// TIA Portal V18 export
TYPE "PLCtoMES_ResultsStoredScanExchange_ext"
// stored: IsFailsafeCompliant false
   STRUCT
      Load_Scanner1ChickInReq : Bool;   // Scanner1查询
      Load_Scanner2ChickInReq : Bool;   // Spare
      Load_Scanner3ChickInReq : Bool;   // Spare
      Load_Scanner4ChickInReq : Bool;   // Spare
      Load_Scanner5ChickInReq : Bool;   // Spare
      Load_Scanner6ChickInReq : Bool;   // Spare
      Load_Scanner7ChickInReq : Bool;   // Spare
      Load_Scanner8ChickInReq : Bool;   // Spare
      SpareByte : Byte;   // Spare
   END_STRUCT;
END_TYPE
